// TIA Portal V17 export
// export: Created 2026-04-13T11:12:04.802365Z, ExportSetting WithDefaults, DisplayName Totally Integrated Automation Portal, DisplayVersion V17 Update 4, DisplayName TIA Portal Openness, DisplayVersion V17 Update 4, DisplayName TIA Portal Version Control Interface, DisplayVersion V17, DisplayName SINAMICS Startdrive Advanced, DisplayVersion V17, DisplayName SINAMICS Startdrive G130, G150, S120, S150, SINAMICS MV, S210, DisplayVersion V17, DisplayName SINAMICS Startdrive G110M, G120, G120C, G120D, G120P, G115D, DisplayVersion V17, DisplayName STEP 7 Professional, DisplayVersion V17 Update 4, DisplayName STEP 7 Safety, DisplayVersion V17, DisplayName WinCC Professional, DisplayVersion V17 Update 4
DATA_BLOCK "BS"   // DB44
{ S7_Optimized_Access := 'TRUE' }
VERSION : 0.1
// stored: AutoNumber true, DBAccessibleFromOPCUA true, DBAccessibleFromWebserver true, IsOnlyStoredInLoadMemory false, IsRetainMemResEnabled false, IsWriteProtectedInAS false, MemoryReserve 100
   VAR RETAIN
      JF进风流量上阈值 : Real := 150.0;
      JF进风流量下阈值 : Real := 150.0;
      ZT主塔压力引风升临界 : Real := 900.0;
      JF进风流量引风关临界 : Real := 2000.0;
      JF进风流量送风关临界 : Real := 1300.0;
      SF送风机1分钟升速 : Real := 4.0;
      YP预喷雾检测主塔压力维持时间 : Int := 30;
      YP预喷雾检测高压 : Real := 800.0;
      YP预喷雾检测低压 : Real := -300.0;
      YP预喷雾检测系统结果 : Int := 1;
      YP预喷雾检测系统正常 : Bool := TRUE;
      YP预喷雾进风流量 : Real := 1500.0;
      "YP预喷雾-离雾-进温" : Real := 100.0;
      "YP预喷雾-离雾-出温" : Real := 85.0;
      YP预喷雾温稳正式时间 : Int := 100;
      GJ关机洗喷头时间 : Int := 60;
      "GJ关机-停水-出温" : Real := 110.0;
      "GJ关机-停水-停雾" : DInt := 60;
      "GJ关机-四参数关-进温" : Real := 70.0;
      "GJ关机-输送-送温" : Real := 65.0;
      ZD自动运行报警 : Bool := FALSE;
      BD步段运行_秒 : Int := 0;
      BD步段运行_分 : Int := 0;
      BD步段运行_时 : Int := 0;
      ZY总运行_秒 : Int := 0;
      ZY总运行_分 : Int := 0;
      ZY总运行_时 : Int := 0;
      JL进料_时 : Int := 0;
      JL进料_分 : Int := 0;
      JL进料_秒 : Int := 0;
      BD步段设定 : Int := 0;
      BD步段运行 : Int := 0;
      ZD自动停止 : Bool := FALSE;
      AQ安全停机 : Bool := FALSE;
      JL进料时间设定 : Real := 10.0;
      XT系统状态 : Int := 1;
      JL进料进风阈值 : Real := 5.0;
      JL进料出风条件 : Real := 80.0;
   END_VAR
   VAR
      WQ尾气温度设定 : Real := 30.0;
      CF出温高报 : Real := 110.0;
      CF出温高高报 : Real := 130.0;
      WQ尾温高报 : Real := 35.0;
      WQ尾温高高报 : Real := 40.0;
      JF进温高报 : Real := 130.0;
      JF进温高高报 : Real := 150.0;
   END_VAR
BEGIN
END_DATA_BLOCK
